TYPE U_INSTANCE_CTRL :
UNION
  stCtrl              : ARRAY[1..MAX_PROCESS] OF ST_INSTANCE_CTRL;
  byCtrl    AT %q*    : ARRAY[1..MAX_PROCESS] OF
                        ARRAY[1..SIZEOF(ST_INSTANCE_CTRL)] OF BYTE;
END_UNION
END_TYPE

(* stored: Version 1.1.0.1
   DUT U_INSTANCE_CTRL: Id {1b3c35d5-a9be-4597-90ea-287dd77e0b12} *)
